TYPE T_OAC_Filename : T_MaxString;
END_TYPE

(* stored: Version 1.1.0.1, ProductVersion 3.1.4024.15
   DUT T_OAC_Filename: Id {96feb316-fec0-4ea1-8b1a-61c26eff22b8} *)
